// TIA Portal V15.1 export
// export: Created 2024-05-17T05:38:44.8004147Z, ExportSetting WithDefaults, DisplayName Totally Integrated Automation Portal, DisplayVersion V15.1 Update 5, DisplayName TIA Portal Openness, DisplayVersion V15.1 Update 5, DisplayName SINAMICS Startdrive Advanced, DisplayVersion V15.1, DisplayName G130, G150, S120, S150, SINAMICS MV, S210, DisplayVersion V15.1, DisplayName G110M, G120, G120C, G120D, G120P, DisplayVersion V15.1, DisplayName STEP 7 Professional, DisplayVersion V15.1 Update 5, DisplayName STEP 7 Safety, DisplayVersion V15.1, DisplayName WinCC Professional, DisplayVersion V15.1 Update 5, DisplayName SIMATIC Visualization Architect, DisplayVersion V15.1
FUNCTION_BLOCK "LGBSoftDet"   // FB6650, FBD
TITLE = LGBSoftDet
{ S7_Optimized_Access := 'FALSE' }
AUTHOR : Imtech
VERSION : 1.0
// stored: AutoNumber false, IsIECCheckEnabled false, SetENOAutomatically False, UDAEnableTagReadback false
   VAR_INPUT
      I_ActualPosition { ExternalAccessible := 'False'; ExternalVisible := 'False'; ExternalWritable := 'False'} : DInt;   // Measuring value comming from the encoder
      C_Position { ExternalAccessible := 'False'; ExternalVisible := 'False'; ExternalWritable := 'False'} : DInt;   // Setpoint position
      C_Diff_HHH_LLL { ExternalAccessible := 'False'; ExternalVisible := 'False'; ExternalWritable := 'False'} : DInt;   // Difference HHH / LLL
      C_Diff_HH_LL { ExternalAccessible := 'False'; ExternalVisible := 'False'; ExternalWritable := 'False'} : DInt;   // Difference HH / LL
      C_Diff_H_L { ExternalAccessible := 'False'; ExternalVisible := 'False'; ExternalWritable := 'False'} : DInt;   // Difference H / L
      C_EnablePos { ExternalAccessible := 'False'; ExternalVisible := 'False'; ExternalWritable := 'False'} : Bool;   // Position is used
   END_VAR
   VAR_OUTPUT
      O_StopHighSpeed { ExternalAccessible := 'False'; ExternalVisible := 'False'; ExternalWritable := 'False'} : Bool;   // Stop high speed
      O_StopLowSpeed { ExternalAccessible := 'False'; ExternalVisible := 'False'; ExternalWritable := 'False'} : Bool;   // Stop low speed
      O_StopPosition { ExternalAccessible := 'False'; ExternalVisible := 'False'; ExternalWritable := 'False'} : Bool;   // Stop on position
      H_IAnim { ExternalAccessible := 'False'; ExternalVisible := 'False'; ExternalWritable := 'False'} : DWord;   // Icon animation
   END_VAR
   VAR_IN_OUT
      H_GBSoftDet : "H_GBSoftDet";   // Animation
   END_VAR
   VAR DB_SPECIFIC
      LevelHHH { ExternalAccessible := 'False'; ExternalVisible := 'False'; ExternalWritable := 'False'} : DInt;   // Level HHH
      LevelHH { ExternalAccessible := 'False'; ExternalVisible := 'False'; ExternalWritable := 'False'} : DInt;   // Level HH
      LevelH { ExternalAccessible := 'False'; ExternalVisible := 'False'; ExternalWritable := 'False'} : DInt;   // Level H
      LevelL { ExternalAccessible := 'False'; ExternalVisible := 'False'; ExternalWritable := 'False'} : DInt;   // Level L
      LevelLL { ExternalAccessible := 'False'; ExternalVisible := 'False'; ExternalWritable := 'False'} : DInt;   // Level LL
      LevelLLL { ExternalAccessible := 'False'; ExternalVisible := 'False'; ExternalWritable := 'False'} : DInt;   // Level LLL
      StopHighSpeed { ExternalAccessible := 'False'; ExternalVisible := 'False'; ExternalWritable := 'False'} : Bool;   // Stop high speed
      StopLowSpeed { ExternalAccessible := 'False'; ExternalVisible := 'False'; ExternalWritable := 'False'} : Bool;   // Stop low speed
      StopPosition { ExternalAccessible := 'False'; ExternalVisible := 'False'; ExternalWritable := 'False'} : Bool;   // Stop on position
   END_VAR
BEGIN

REGION Network 1: **** 4.6 - Machine Status - Indication **** Icon Animation
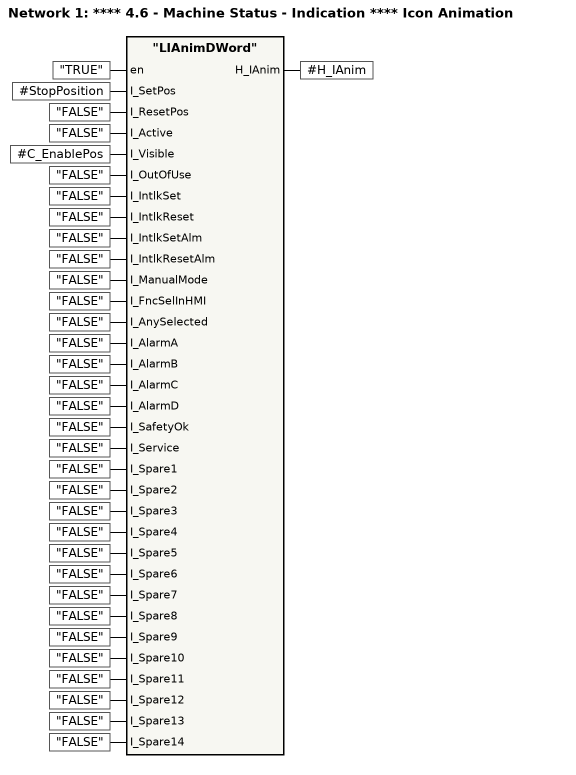
   IF "TRUE" THEN
       "LIAnimDWord"(I_SetPos := #StopPosition,
                     I_ResetPos := "FALSE",
                     I_Active := "FALSE",
                     I_Visible := #C_EnablePos,
                     I_OutOfUse := "FALSE",
                     I_IntlkSet := "FALSE",
                     I_IntlkReset := "FALSE",
                     I_IntlkSetAlm := "FALSE",
                     I_IntlkResetAlm := "FALSE",
                     I_ManualMode := "FALSE",
                     I_FncSelInHMI := "FALSE",
                     I_AnySelected := "FALSE",
                     I_AlarmA := "FALSE",
                     I_AlarmB := "FALSE",
                     I_AlarmC := "FALSE",
                     I_AlarmD := "FALSE",
                     I_SafetyOk := "FALSE",
                     I_Service := "FALSE",
                     I_Spare1 := "FALSE",
                     I_Spare2 := "FALSE",
                     I_Spare3 := "FALSE",
                     I_Spare4 := "FALSE",
                     I_Spare5 := "FALSE",
                     I_Spare6 := "FALSE",
                     I_Spare7 := "FALSE",
                     I_Spare8 := "FALSE",
                     I_Spare9 := "FALSE",
                     I_Spare10 := "FALSE",
                     I_Spare11 := "FALSE",
                     I_Spare12 := "FALSE",
                     I_Spare13 := "FALSE",
                     I_Spare14 := "FALSE",
                     H_IAnim => #H_IAnim);
   END_IF;
END_REGION

REGION Network 2: **** 4.6 - Machine Status - Indications **** Animation
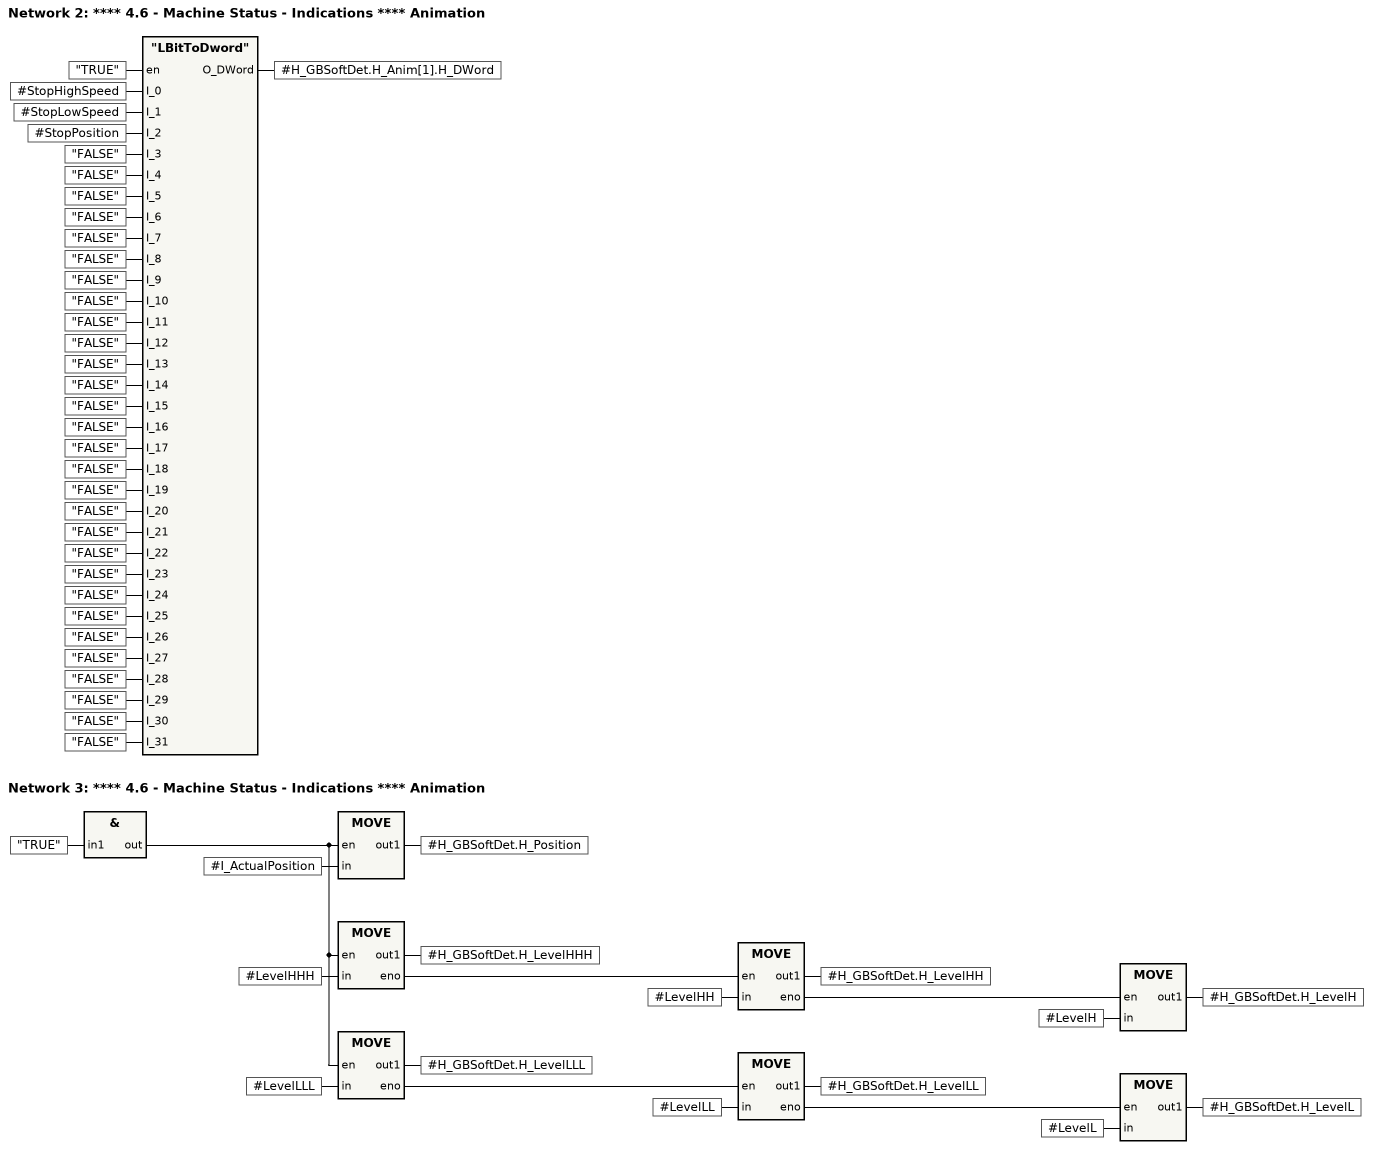
   IF "TRUE" THEN
       "LBitToDword"(I_0 := #StopHighSpeed,
                     I_1 := #StopLowSpeed,
                     I_2 := #StopPosition,
                     I_3 := "FALSE",
                     I_4 := "FALSE",
                     I_5 := "FALSE",
                     I_6 := "FALSE",
                     I_7 := "FALSE",
                     I_8 := "FALSE",
                     I_9 := "FALSE",
                     I_10 := "FALSE",
                     I_11 := "FALSE",
                     I_12 := "FALSE",
                     I_13 := "FALSE",
                     I_14 := "FALSE",
                     I_15 := "FALSE",
                     I_16 := "FALSE",
                     I_17 := "FALSE",
                     I_18 := "FALSE",
                     I_19 := "FALSE",
                     I_20 := "FALSE",
                     I_21 := "FALSE",
                     I_22 := "FALSE",
                     I_23 := "FALSE",
                     I_24 := "FALSE",
                     I_25 := "FALSE",
                     I_26 := "FALSE",
                     I_27 := "FALSE",
                     I_28 := "FALSE",
                     I_29 := "FALSE",
                     I_30 := "FALSE",
                     I_31 := "FALSE",
                     O_DWord => #H_GBSoftDet.H_Anim[1].H_DWord);
   END_IF;
END_REGION

REGION Network 3: **** 4.6 - Machine Status - Indications **** Animation
   IF "TRUE" THEN
       #H_GBSoftDet.H_Position := #I_ActualPosition;
       #H_GBSoftDet.H_LevelHHH := #LevelHHH;
       #H_GBSoftDet.H_LevelHH := #LevelHH;
       #H_GBSoftDet.H_LevelH := #LevelH;
       #H_GBSoftDet.H_LevelLLL := #LevelLLL;
       #H_GBSoftDet.H_LevelLL := #LevelLL;
       #H_GBSoftDet.H_LevelL := #LevelL;
   END_IF;
END_REGION

REGION Network 4: **** 5.2 - Equations - Equations **** Level LLL
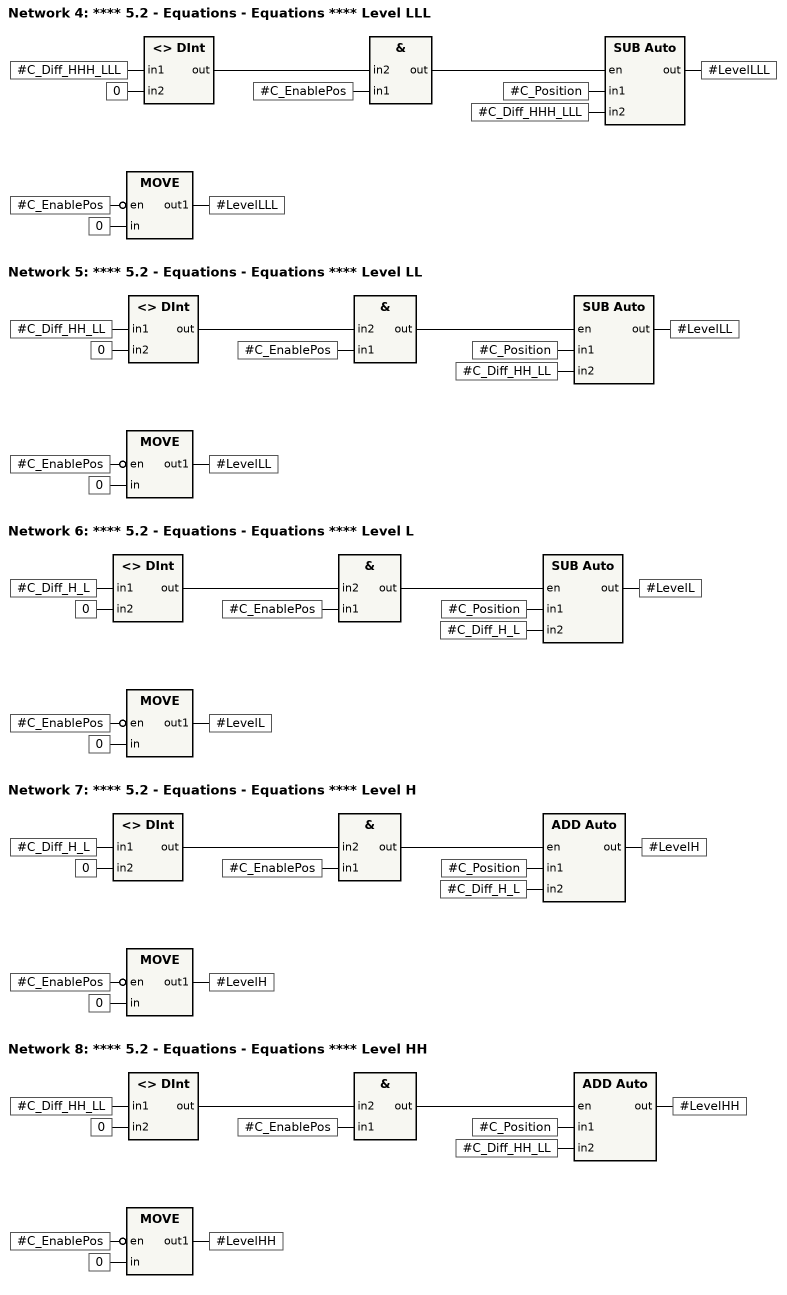
   IF (#C_Diff_HHH_LLL <> 0) AND #C_EnablePos THEN #LevelLLL := #C_Position - #C_Diff_HHH_LLL; END_IF;
   IF NOT #C_EnablePos THEN #LevelLLL := 0; END_IF;
END_REGION

REGION Network 5: **** 5.2 - Equations - Equations **** Level LL
   IF (#C_Diff_HH_LL <> 0) AND #C_EnablePos THEN #LevelLL := #C_Position - #C_Diff_HH_LL; END_IF;
   IF NOT #C_EnablePos THEN #LevelLL := 0; END_IF;
END_REGION

REGION Network 6: **** 5.2 - Equations - Equations **** Level L
   IF (#C_Diff_H_L <> 0) AND #C_EnablePos THEN #LevelL := #C_Position - #C_Diff_H_L; END_IF;
   IF NOT #C_EnablePos THEN #LevelL := 0; END_IF;
END_REGION

REGION Network 7: **** 5.2 - Equations - Equations **** Level H
   IF (#C_Diff_H_L <> 0) AND #C_EnablePos THEN #LevelH := #C_Position + #C_Diff_H_L; END_IF;
   IF NOT #C_EnablePos THEN #LevelH := 0; END_IF;
END_REGION

REGION Network 8: **** 5.2 - Equations - Equations **** Level HH
   IF (#C_Diff_HH_LL <> 0) AND #C_EnablePos THEN #LevelHH := #C_Position + #C_Diff_HH_LL; END_IF;
   IF NOT #C_EnablePos THEN #LevelHH := 0; END_IF;
END_REGION

REGION Network 9: **** 5.2 - Equations - Equations **** Level HHH
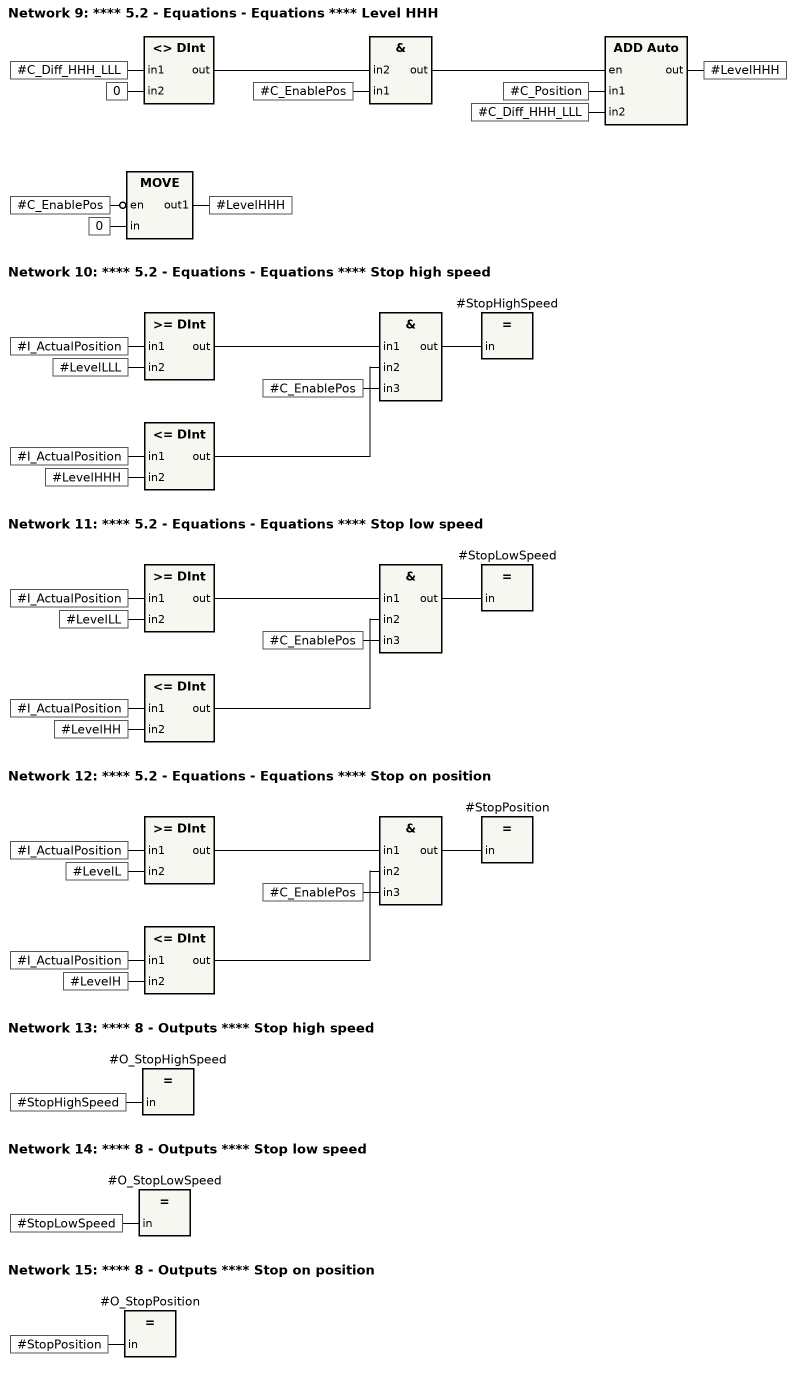
   IF (#C_Diff_HHH_LLL <> 0) AND #C_EnablePos THEN #LevelHHH := #C_Position + #C_Diff_HHH_LLL; END_IF;
   IF NOT #C_EnablePos THEN #LevelHHH := 0; END_IF;
END_REGION

REGION Network 10: **** 5.2 - Equations - Equations **** Stop high speed
   #StopHighSpeed := (#I_ActualPosition >= #LevelLLL) AND (#I_ActualPosition <= #LevelHHH) AND #C_EnablePos;
END_REGION

REGION Network 11: **** 5.2 - Equations - Equations **** Stop low speed
   #StopLowSpeed := (#I_ActualPosition >= #LevelLL) AND (#I_ActualPosition <= #LevelHH) AND #C_EnablePos;
END_REGION

REGION Network 12: **** 5.2 - Equations - Equations **** Stop on position
   #StopPosition := (#I_ActualPosition >= #LevelL) AND (#I_ActualPosition <= #LevelH) AND #C_EnablePos;
END_REGION

REGION Network 13: **** 8 - Outputs **** Stop high speed
   #O_StopHighSpeed := #StopHighSpeed;
END_REGION

REGION Network 14: **** 8 - Outputs **** Stop low speed
   #O_StopLowSpeed := #StopLowSpeed;
END_REGION

REGION Network 15: **** 8 - Outputs **** Stop on position
   #O_StopPosition := #StopPosition;
END_REGION
END_FUNCTION_BLOCK
